{attribute 'GeneratedUsingTerminal: EP9576-1032-0016'}
{attribute addProperty BoxType "EP9576-1032-0016"}
{attribute addProperty Id "BCT_InputsAT %I*BCT_Inputs_7ACE8FA617WcStateAT %I*WcState_9091E0EB2InfoDataAT %I*InfoData_32EB74EA10"}
{attribute addProperty CRC "3290514118"}
{attribute addProperty Size "29"}
TYPE EP9576_C42142C6 EXTENDS EtcSlaveTerminalBase_947E5A46 :
STRUCT
	{attribute addProperty Name "BCT_Inputs"}
	BCT_Inputs : BCT_Inputs_7ACE8FA6;
	{attribute addProperty Name "WcState"}
	WcState : WcState_9091E0EB;
	{attribute addProperty Name "InfoData"}
	InfoData : InfoData_32EB74EA;
END_STRUCT
END_TYPE

(* stored: Version 1.2.0.0, ProductVersion 3.1.4024.9
   DUT EP9576_C42142C6: Id {0c31fd44-aa88-4a30-9f91-2243d481dd52} *)
